// TIA Portal V20 export
DATA_BLOCK "DB_Manual"   // DB22
// stored: Access Published, MemoryReserve 100, Namespace Global
   VAR
      Conveyor : Struct
         ID : Int;
         Enable : Bool;
         Run : Bool;
         in : Bool;
      END_STRUCT;
      Line : Struct
         ProductionLine : Struct
            Conveyor { S7_SetPoint := 'True'} : Array[_.gminProductionLine.._.gmaxProductionLine] of "Global.ManualInputs";
         END_STRUCT;
         EmptyLine : Struct
            Conveyor { S7_SetPoint := 'True'} : Array[_.gminEmptyLine.._.gmaxEmptyLine] of "Global.ManualInputs";
         END_STRUCT;
         PackedLine : Struct
            Conveyor { S7_SetPoint := 'True'} : Array[_.gminPackedLine.._.gmaxPackedLine] of "Global.ManualInputs";
         END_STRUCT;
      END_STRUCT;
   END_VAR
BEGIN
END_DATA_BLOCK
